FUNCTION_BLOCK FB_Descargar_SFC

VAR_INPUT
    // SFC-Flags
    SFCPause: BOOL;
    SFCReset: BOOL;
    
	// Sincronizacion
    Benido: BOOL ;
    Ejecuta: BOOL;
    
	// Parametros de control de la estacion
    //CicloACiclo: BOOL;    
    DescargadorDetras AT %I* : BOOL;
    DescargadorDelante AT %I* : BOOL;
    DescargadorArriba AT %I* : BOOL;
    DescargadorAbajo AT %I* : BOOL;
END_VAR
VAR_OUTPUT
   // DescargadorAvanza AT %Q* : BOOL;
   // DescargadorBaja AT %Q* : BOOL;
   // DescargadorCierra AT %Q* : BOOL;
    DescargadorAvanza: BOOL;
    DescargadorBaja: BOOL;
    DescargadorCierra: BOOL;

	// Sincronizacion    
    Acabhe: BOOL;
    ListoKalisto: BOOL;
END_VAR

VAR_IN_OUT
	    cont: UINT;
END_VAR

VAR
END_VAR

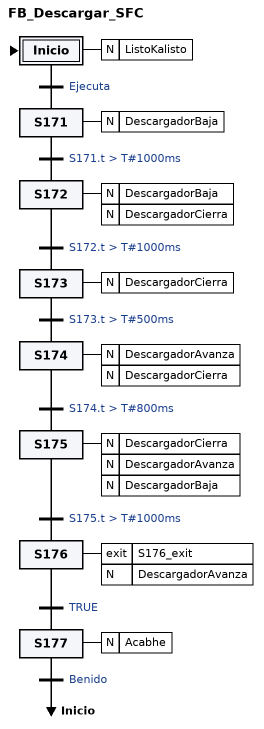
INITIAL_STEP Inicio:
    ListoKalisto(N);
END_STEP
TRANSITION FROM Inicio TO S171
    := Ejecuta;
END_TRANSITION
STEP S171:
    DescargadorBaja(N);
END_STEP
TRANSITION FROM S171 TO S172
    := S171.t > T#1000ms;
END_TRANSITION
STEP S172:
    DescargadorBaja(N);
    DescargadorCierra(N);
END_STEP
TRANSITION FROM S172 TO S173
    := S172.t > T#1000ms;
END_TRANSITION
STEP S173:
    DescargadorCierra(N);
END_STEP
TRANSITION FROM S173 TO S174
    := S173.t > T#500ms;
END_TRANSITION
STEP S174:
    DescargadorAvanza(N);
    DescargadorCierra(N);
END_STEP
TRANSITION FROM S174 TO S175
    := S174.t > T#800ms;
END_TRANSITION
STEP S175:
    DescargadorCierra(N);
    DescargadorAvanza(N);
    DescargadorBaja(N);
END_STEP
TRANSITION FROM S175 TO S176
    := S175.t > T#1000ms;
END_TRANSITION
STEP S176:
    S176_exit(P0);  // exit action
    DescargadorAvanza(N);
END_STEP
TRANSITION FROM S176 TO S177
    := TRUE;
END_TRANSITION
STEP S177:
    Acabhe(N);
END_STEP
TRANSITION FROM S177 TO Inicio
    := Benido;
END_TRANSITION

ACTION S176_exit:
cont := cont + 1;
END_ACTION

END_FUNCTION_BLOCK

(* stored: Version 1.1.0.1, ProductVersion 3.1.4024.12
   POU FB_Descargar_SFC: Id {eb449dff-be2f-474e-9f3e-38c4f991f01b}, SpecialFunc None
   Action S176_exit: Id {04f0c0d5-f241-4c8a-a5e2-369a15e67f08} *)
